FUNCTION_BLOCK EL1899
VAR
	_io : EL1xx9_Data;
	{attribute addProperty Name "WcState"}
	_wcState : WcStateInputToggle;
	{attribute addProperty Name "Info data"}
	_infoData : InfoDataBase;
END_VAR

PROPERTY IO : REFERENCE TO EL1xx9_Data
GET
IO REF= _io;
END_GET
END_PROPERTY

PROPERTY WcState : REFERENCE TO WcStateInputToggle
GET
WcState REF= _wcState;
END_GET
END_PROPERTY

END_FUNCTION_BLOCK

(* stored: Version 1.1.0.1, ProductVersion 3.1.4024.9
   POU EL1899: Id {f869e664-bf85-05fb-3d90-2c0343154a7c}, SpecialFunc None
   Property IO: Id {8dcfb8cc-dfd6-0965-064a-79412a07523b}
   Get Get: Id {dd1c4d0c-5018-03c1-0e03-07c6a2f392fd}
   Property WcState: Id {0c159500-ea33-0889-3f9e-593c87908bb4}
   Get Get: Id {38cf1ad2-55c9-068c-3582-ab32f6ddeaa5} *)
